INTERFACE I_PersistentEventStorage

METHOD StoreEvent
VAR_INPUT
	stEvent : ST_Event;
END_VAR
END_METHOD

END_INTERFACE

(* stored: Version 1.1.0.1, ProductVersion 3.1.4024.12
   Itf I_PersistentEventStorage: Id {bc628b9f-34af-4757-bcba-8c2fa3a014b0}
   Method StoreEvent: Id {25228aa2-ab10-404f-8764-597ee37dd627} *)
